ADAPTER IORevPiBusAdapter (* Bus Adapter for Revolution Pi by KUNBUS GmbH *)
  (* Standard: 61499-2; Description: Copyright (c) 2018 fortiss GmbH This program and the accompanying materials are made available under the terms of the Eclipse Public License 2.0 which is available at https://www.eclipse.org/legal/epl-2.0/ SPDX-License-Identifier: EPL-2.0 *)
  (* Version 1.0, 2018-04-22, José Cabral, fortiss GmbH *)
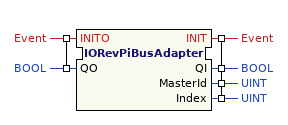
  EVENT_INPUT
    INITO WITH QO; (* Initialization Confirm *)
  END_EVENT
  EVENT_OUTPUT
    INIT WITH Index, MasterId, QI; (* Service Initialization *)
  END_EVENT
  VAR_INPUT
    QO : BOOL;
  END_VAR
  VAR_OUTPUT
    QI : BOOL;
    MasterId : UINT;
    Index : UINT;
  END_VAR
  SERVICE SOCKET/PLUG (* Bus Adapter for Revolution Pi by KUNBUS GmbH *)
    SEQUENCE request_confirm
      SOCKET.REQ(REQD) -> PLUG.REQ(REQD);
      PLUG.CNF(CNFD) -> SOCKET.CNF(CNFD);
    END_SEQUENCE
    SEQUENCE indication_response
      PLUG.IND(INDD) -> SOCKET.IND(INDD);
      SOCKET.RSP(RSPD) -> PLUG.RSP(RSPD);
    END_SEQUENCE
  END_SERVICE
END_ADAPTER
